% RSLogix 500 project Mackerel_Deck.RSS, saved by version 8.30.00.16 %
PROJECT "DECK"    % processor: Bul.1763 MicroLogix 1100 Series B %

PROGRAM FILES
  LAD 2   7 rungs

DATA FILES
  O0 OUTPUT  8 elements
  I1 INPUT  14 elements
  S2 STATUS  66 elements
  B3 BINARY  1 elements
  T4 TIMER  2 elements
  C5 COUNTER  1 elements
  R6 CONTROL  1 elements
  N7 INTEGER  2 elements
  F8 FLOAT  1 elements

LADDER 2
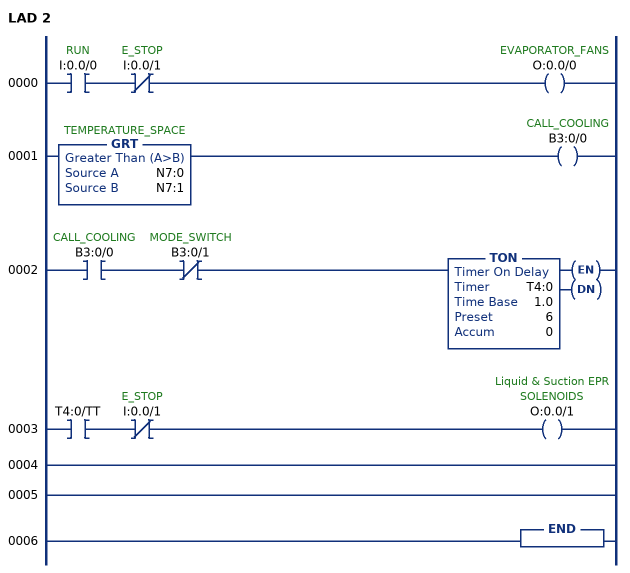
% Rung: 0 %
SOR XIC I:0.0/0 XIO I:0.0/1 OTE O:0.0/0 EOR
%   I:0.0/0  RUN %
%   I:0.0/1  E_STOP %
%   O:0.0/0  EVAPORATOR_FANS %
% Rung: 1 %
SOR GRT N7:0 N7:1 OTE B3:0/0 EOR
%   N7:0  TEMPERATURE_SPACE %
%   N7:1  TEMPERTURE_SET_POINT %
%   B3:0/0  CALL_COOLING %
% Rung: 2 %
SOR XIC B3:0/0 XIO B3:0/1 TON T4:0 1.0 6 0 EOR
%   B3:0/0  CALL_COOLING %
%   B3:0/1  MODE_SWITCH %
% Rung: 3 %  % edit flag set %
SOR XIC T4:0/TT XIO I:0.0/1 OTE O:0.0/1 EOR
%   I:0.0/1  E_STOP %
%   O:0.0/1  SOLENOIDS  "Liquid & Suction EPR" %
% Rung: 4 %  % edit flag set %
SOR EOR
% Rung: 5 %  % edit flag set %
SOR EOR
% Rung: 6 %
SOR END EOR

OTHER DOCUMENTED ADDRESSES
  T4:0/0  MODE_COOLING_ON

REVISION NOTES
  0: Switch for fans.
  1: Compiled?
  2: Able to affect emulation.
  3: Run/E-stop
  4: Emulator?
  5: E-stop

DATA TABLE (non-zero values as saved)
DATA T4
% .PRE .ACC %
% T4:0 % 6 0
DATA N7
% N7:0 % 46 44
